SYSTEM test
  (* Version 1.0, 2022-12-08, franz *)
  APPLICATION testApp
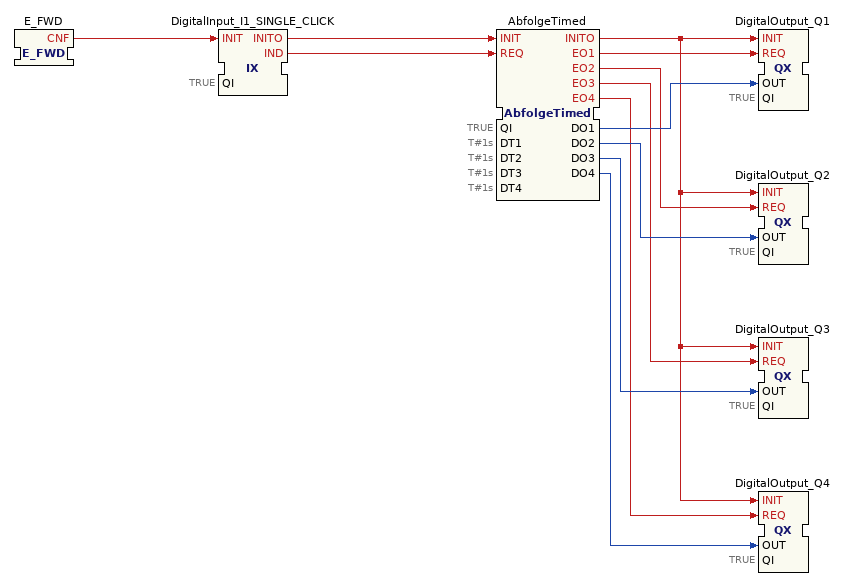
    FBS
      DigitalInput_I1_SINGLE_CLICK : IX(QI := TRUE);
      DigitalOutput_Q1 : QX(QI := TRUE);
      E_FWD : E_FWD;
      DigitalOutput_Q2 : QX(QI := TRUE);
      DigitalOutput_Q3 : QX(QI := TRUE);
      DigitalOutput_Q4 : QX(QI := TRUE);
      AbfolgeTimed : AbfolgeTimed(QI := TRUE, DT1 := T#1s, DT2 := T#1s, DT3 := T#1s, DT4 := T#1s);
    END_FBS
    EVENT_CONNECTIONS
      E_FWD.CNF TO DigitalInput_I1_SINGLE_CLICK.INIT;
      DigitalInput_I1_SINGLE_CLICK.INITO TO AbfolgeTimed.INIT;
      DigitalInput_I1_SINGLE_CLICK.IND TO AbfolgeTimed.REQ;
      AbfolgeTimed.INITO TO DigitalOutput_Q1.INIT;
      AbfolgeTimed.INITO TO DigitalOutput_Q2.INIT;
      AbfolgeTimed.INITO TO DigitalOutput_Q3.INIT;
      AbfolgeTimed.INITO TO DigitalOutput_Q4.INIT;
      AbfolgeTimed.EO1 TO DigitalOutput_Q1.REQ;
      AbfolgeTimed.EO2 TO DigitalOutput_Q2.REQ;
      AbfolgeTimed.EO3 TO DigitalOutput_Q3.REQ;
      AbfolgeTimed.EO4 TO DigitalOutput_Q4.REQ;
    END_CONNECTIONS
    DATA_CONNECTIONS
      AbfolgeTimed.DO1 TO DigitalOutput_Q1.OUT;
      AbfolgeTimed.DO2 TO DigitalOutput_Q2.OUT;
      AbfolgeTimed.DO3 TO DigitalOutput_Q3.OUT;
      AbfolgeTimed.DO4 TO DigitalOutput_Q4.OUT;
    END_CONNECTIONS
  END_APPLICATION
  APPLICATION mapping
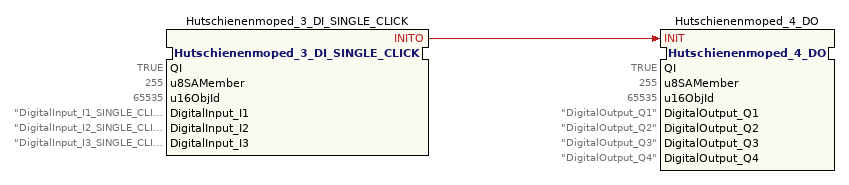
    FBS
      Hutschienenmoped_3_DI_SINGLE_CLICK : Hutschienenmoped_3_DI_SINGLE_CLICK(QI := TRUE, u8SAMember := 255, u16ObjId := 65535, DigitalInput_I1 := "DigitalInput_I1_SINGLE_CLICK", DigitalInput_I2 := "DigitalInput_I2_SINGLE_CLICK", DigitalInput_I3 := "DigitalInput_I3_SINGLE_CLICK");
      Hutschienenmoped_4_DO : Hutschienenmoped_4_DO(QI := TRUE, u8SAMember := 255, u16ObjId := 65535, DigitalOutput_Q1 := "DigitalOutput_Q1", DigitalOutput_Q2 := "DigitalOutput_Q2", DigitalOutput_Q3 := "DigitalOutput_Q3", DigitalOutput_Q4 := "DigitalOutput_Q4");
    END_FBS
    EVENT_CONNECTIONS
      Hutschienenmoped_3_DI_SINGLE_CLICK.INITO TO Hutschienenmoped_4_DO.INIT;
    END_CONNECTIONS
  END_APPLICATION
  DEVICE FORTE_PC : FORTE_PC(MGR_ID := "192.168.4.1:61499")
    {SET_ATTRIBUTE(Profile, DynamicTypeLoad)}
    {SET_ATTRIBUTE(FBType, GEN_E_MUX, F_LT, E_CTD, E_STOPWATCH, F_LIMIT, UT_AuxiliaryInputMapping, UT_ButtonMapping_UP, F_TIME_IN_S_TO_UDINT, F_TAN, Hutschienenmoped_6_DIA_LONG_PRESS_START, Hutschienenmoped_3_DI_LONG_PRESS_START, COLOR_BLACK, F_ACOS, QD, COLOR_WHITE, COLOR_OLIVE, E_MERGE, Hutschienenmoped_3_DI_DOUBLE_CLICK, EMB_RES, COLOR_CYAN, ID, E_DEMUX, NVS_UDINT, AbfolgeTipp, GEN_SUBL, Hutschienenmoped_6_DIA_LONG_PRESS_HOLD, QW, QX, F_MUL, IW, IX, Q_ChangePolygonScale, F_LE, GEN_SUBSCRIBE, Hutschienenmoped_3_DI_SINGLE_CLICK, F_ATAN, Hutschienenmoped_3_DI, GEN_AND, F_SIN, F_LN, GEN_CLIENT, F_NOT, COLOR_MAROON, GEN_SERVER, GEN_PUBL, Q_SelectActiveWorkingSet, RMT_RES, COLOR_RED, UT_ButtonMapping_HOLD, GEN_OR, E_D_FF, Hutschienenmoped_6_DIA_DOUBLE_CLICK, E_CYCLE, UT_ButtonMapping, E_R_TRIG, COLOR_TEAL, COLOR_BLUE, Q_ActiveMask, F_GE, E_F_TRIG, E_RS, F_MUX_2, DEV_MGR, E_SPLIT, E_FWD, E_CTUD, UT_SoftkeyMapping_UP, F_EQ, E_T_FF, E_RDELAY, UT_ButtonMapping_DOWN, F_MOD, E_RTimeOut, F_NE, Hutschienenmoped_6_DIA_REPEAT, NVS_UINT, Hutschienenmoped_3_DI_UP, CbVtStatus, Q_ObjEnableDisable, F_TIME_IN_NS_TO_UDINT, FB_RANDOM, F_EXP, E_SELECT, GEN_PUBLISH, Hutschienenmoped_4_DO, Hutschienenmoped_6_DIA, F_TIME_IN_MS_TO_UDINT, Hutschienenmoped_6_DIA_SINGLE_CLICK, Hutschienenmoped_3_DI_DOWN, E_CTUD_UDINT, Q_CtrlAudioSignal, E_TRAIN, OUT_ANY_CONSOLE, F_SUB, Q_ChangeObjectLabel, F_GT, COLOR_YELLOW, GEN_E_DEMUX, F_LOG, F_SQRT, E_SR, COLOR_NAVY, GEN_XOR, Q_ChildLocation, F_MIN, Hutschienenmoped_6_DIA_UP, Hutschienenmoped_6_DIA_DOWN, E_SWITCH, E_RESTART, E_PERMIT, UT_SoftkeyMapping_HOLD, F_SEL, Q_ChangePolygonPoint, UT_SoftkeyMapping, F_MAX, E_TimeOut, COLOR_SILVER, Q_BackgroundColour, COLOR_MAGENTA, UT_SoftkeyMapping_DOWN, Q_Attribute, COLOR_LIME, COLOR_GREEN, COLOR_GREY, COLOR_PURPLE, Hutschienenmoped_3_DI_LONG_PRESS_HOLD, F_ABS, E_DELAY, GEN_ADD, F_COS, Q_ObjHideShow, Q_StringValue, F_TIME_IN_US_TO_UDINT, E_CTU, Q_NumericValue, Q_ChildPosition, strip_set_pixel, hsv2rgb, Hutschienenmoped_3_DI_REPEAT, E_REND, F_ASIN, F_DIV)} (* created during deployment *)
    {SET_ATTRIBUTE(AdapterType, ATimeOut, ARTimeOut, ANY_ADAPTER)} (* created during deployment *)
    RESOURCE EMB_RES : EMB_RES
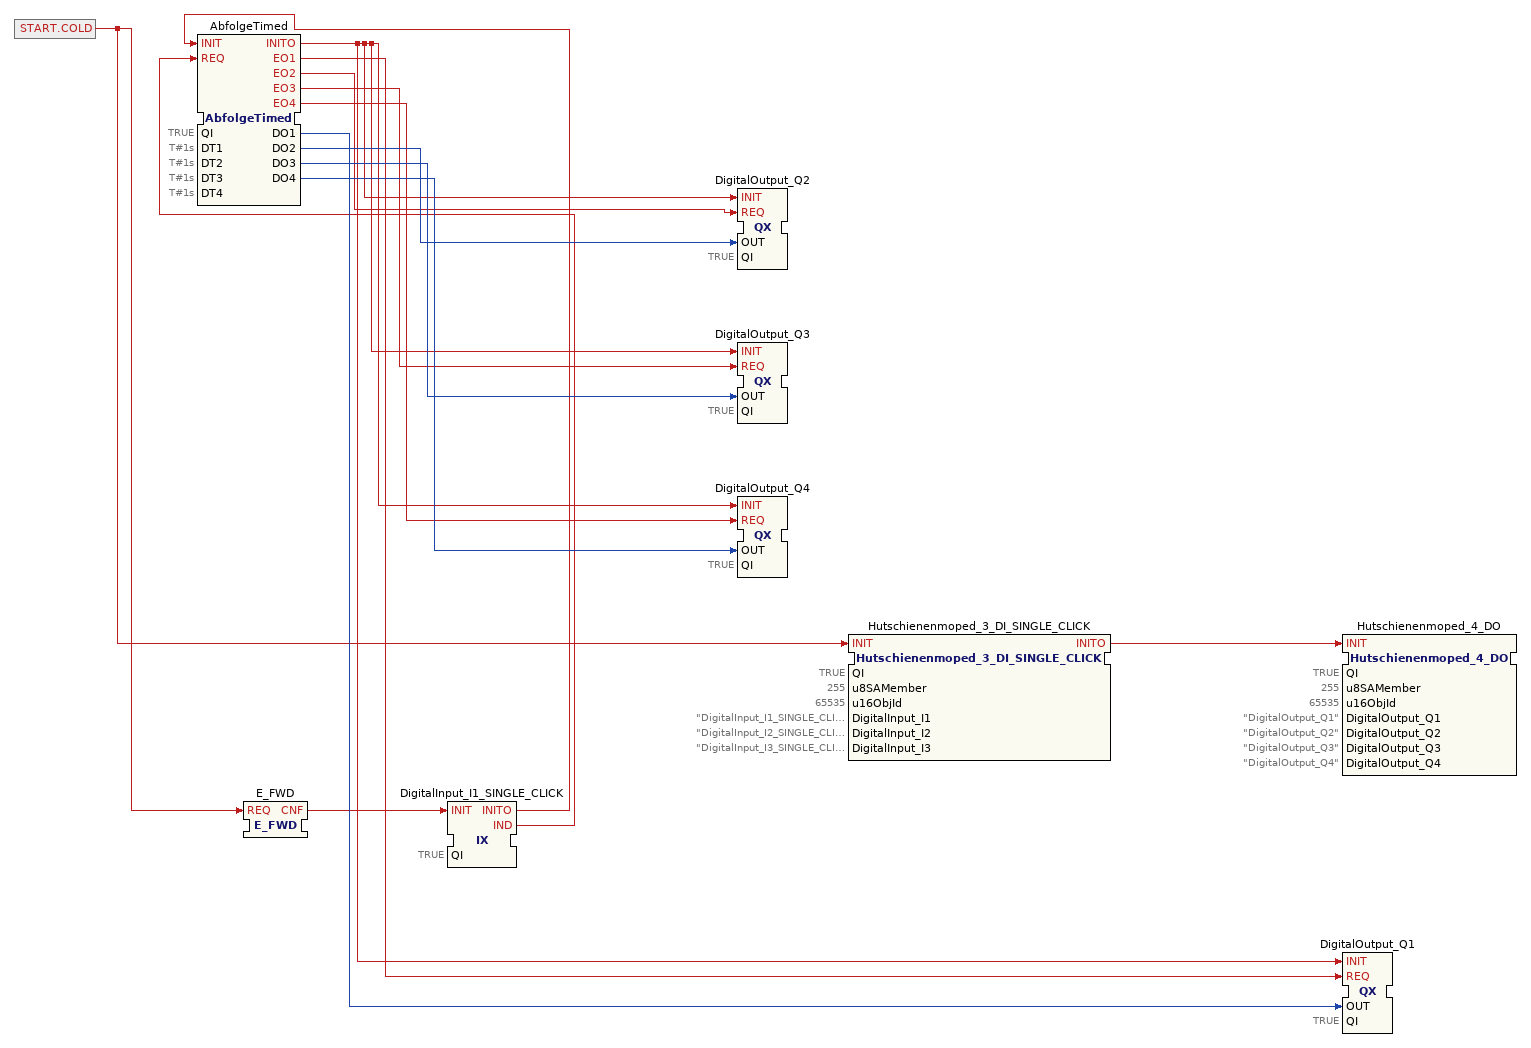
      FBS
        Hutschienenmoped_4_DO : Hutschienenmoped_4_DO(QI := TRUE, u8SAMember := 255, u16ObjId := 65535, DigitalOutput_Q1 := "DigitalOutput_Q1", DigitalOutput_Q2 := "DigitalOutput_Q2", DigitalOutput_Q3 := "DigitalOutput_Q3", DigitalOutput_Q4 := "DigitalOutput_Q4");
        Hutschienenmoped_3_DI_SINGLE_CLICK : Hutschienenmoped_3_DI_SINGLE_CLICK(QI := TRUE, u8SAMember := 255, u16ObjId := 65535, DigitalInput_I1 := "DigitalInput_I1_SINGLE_CLICK", DigitalInput_I2 := "DigitalInput_I2_SINGLE_CLICK", DigitalInput_I3 := "DigitalInput_I3_SINGLE_CLICK");
        DigitalOutput_Q1 : QX(QI := TRUE);
        E_FWD : E_FWD;
        DigitalInput_I1_SINGLE_CLICK : IX(QI := TRUE);
        DigitalOutput_Q2 : QX(QI := TRUE);
        DigitalOutput_Q3 : QX(QI := TRUE);
        DigitalOutput_Q4 : QX(QI := TRUE);
        AbfolgeTimed : AbfolgeTimed(QI := TRUE, DT1 := T#1s, DT2 := T#1s, DT3 := T#1s, DT4 := T#1s);
      END_FBS
      EVENT_CONNECTIONS
        Hutschienenmoped_3_DI_SINGLE_CLICK.INITO TO Hutschienenmoped_4_DO.INIT;
        START.COLD TO Hutschienenmoped_3_DI_SINGLE_CLICK.INIT;
        E_FWD.CNF TO DigitalInput_I1_SINGLE_CLICK.INIT;
        START.COLD TO E_FWD.REQ;
        DigitalInput_I1_SINGLE_CLICK.INITO TO AbfolgeTimed.INIT;
        DigitalInput_I1_SINGLE_CLICK.IND TO AbfolgeTimed.REQ;
        AbfolgeTimed.INITO TO DigitalOutput_Q1.INIT;
        AbfolgeTimed.INITO TO DigitalOutput_Q2.INIT;
        AbfolgeTimed.INITO TO DigitalOutput_Q3.INIT;
        AbfolgeTimed.INITO TO DigitalOutput_Q4.INIT;
        AbfolgeTimed.EO1 TO DigitalOutput_Q1.REQ;
        AbfolgeTimed.EO2 TO DigitalOutput_Q2.REQ;
        AbfolgeTimed.EO3 TO DigitalOutput_Q3.REQ;
        AbfolgeTimed.EO4 TO DigitalOutput_Q4.REQ;
      END_CONNECTIONS
      DATA_CONNECTIONS
        AbfolgeTimed.DO1 TO DigitalOutput_Q1.OUT;
        AbfolgeTimed.DO2 TO DigitalOutput_Q2.OUT;
        AbfolgeTimed.DO3 TO DigitalOutput_Q3.OUT;
        AbfolgeTimed.DO4 TO DigitalOutput_Q4.OUT;
      END_CONNECTIONS
    END_RESOURCE
  END_DEVICE
  MAPPINGS
    mapping.Hutschienenmoped_4_DO ON FORTE_PC.EMB_RES.Hutschienenmoped_4_DO;
    mapping.Hutschienenmoped_3_DI_SINGLE_CLICK ON FORTE_PC.EMB_RES.Hutschienenmoped_3_DI_SINGLE_CLICK;
    testApp.DigitalOutput_Q1 ON FORTE_PC.EMB_RES.DigitalOutput_Q1;
    testApp.E_FWD ON FORTE_PC.EMB_RES.E_FWD;
    testApp.DigitalInput_I1_SINGLE_CLICK ON FORTE_PC.EMB_RES.DigitalInput_I1_SINGLE_CLICK;
    testApp.DigitalOutput_Q2 ON FORTE_PC.EMB_RES.DigitalOutput_Q2;
    testApp.DigitalOutput_Q3 ON FORTE_PC.EMB_RES.DigitalOutput_Q3;
    testApp.DigitalOutput_Q4 ON FORTE_PC.EMB_RES.DigitalOutput_Q4;
    testApp.AbfolgeTimed ON FORTE_PC.EMB_RES.AbfolgeTimed;
  END_MAPPINGS
  SEGMENTS
    Ethernet : Ethernet;
  END_SEGMENTS
  LINKS
    FORTE_PC => Ethernet;
  END_LINKS
END_SYSTEM
